{attribute 'linkalways'} 
{attribute 'no_explicit_call' := 'This FB is a CLASS and must be accessed using methods or properties'}
{attribute 'enable_dynamic_creation'}
FUNCTION_BLOCK _TcVnVector2_UINT EXTENDS AliasDatatypeBase
VAR
	localData : TcVnVector2_UINT;
	activeData : REFERENCE TO TcVnVector2_UINT REF= localData;
	aliasBaseDatatype : _Array0to1OfUINT;
END_VAR

PROPERTY PUBLIC Address : PVOID
GET
Address := ADR(activeData);
END_GET
END_PROPERTY

METHOD PUBLIC ClearReference
VAR_INPUT
END_VAR
activeData REF= localData;
SetBaseDatatypeReference();
END_METHOD

METHOD PUBLIC Clone : I_Datatype
VAR
    pClone : POINTER TO _TcVnVector2_UINT;
END_VAR
pClone := __NEW(_TcVnVector2_UINT);
Clone := pClone^;
END_METHOD

METHOD FB_init : BOOL
VAR_INPUT
	bInitRetains : BOOL; // if TRUE, the retain variables are initialized (warm start / cold start)
	bInCopyCode : BOOL;  // if TRUE, the instance afterwards gets moved into the copy code (online change)
	//InitialValue : <type>; // if possible, not all values can be initialized
END_VAR
//localData := InitialValue; // if possible, not all values can be initialized
SetBaseDatatypeReference();
AddBaseDatatype(aliasBaseDatatype);
END_METHOD

PROPERTY PUBLIC Identifier : T_MAXSTRING
GET
Identifier := 'TcVnVector2_UINT';
END_GET
END_PROPERTY

METHOD PUBLIC MakeReferenceTo
VAR_INPUT
	ReferenceTarget : REFERENCE TO TcVnVector2_UINT;
END_VAR
activeData REF= ReferenceTarget;
SetBaseDatatypeReference();
END_METHOD

METHOD PROTECTED SetBaseDatatypeReference
VAR_INPUT
END_VAR
aliasBaseDatatype.MakeReferenceTo(activeData);
END_METHOD

PROPERTY PUBLIC Size : UDINT
GET
Size := SIZEOF(activeData);
END_GET
END_PROPERTY

METHOD TryMakeReferenceTo : BOOL
VAR_INPUT
	Target : I_Datatype;
END_VAR
VAR
	pTargetData : POINTER TO TcVnVector2_UINT;
END_VAR
IF NOT IsEquivalentTo(Target) THEN
	RETURN;
END_IF

pTargetData := Target.Address;
activeData REF= pTargetData^;
SetBaseDatatypeReference();
TryMakeReferenceTo := TRUE;
END_METHOD

PROPERTY PUBLIC Value : REFERENCE TO TcVnVector2_UINT
GET
Value REF= activeData;
END_GET
END_PROPERTY

END_FUNCTION_BLOCK

(* stored: Version 1.1.0.1, ProductVersion 3.1.4024.13
   POU _TcVnVector2_UINT: Id {8bdec0e3-bc1d-03c1-31a8-aad19038b9a6}, SpecialFunc None
   Folder Core: Id {6b5e70ee-943d-0e8f-172c-51f2530f36c3}
   Folder Protected: Id {119f0d77-7c6b-089f-3a92-8e4dc8a1e82c}
   Folder Customize: Id {2d9d9cb3-6aec-0103-3f2c-dbef9294f431}
   Folder Constructor: Id {b36db007-e1b4-09c8-3b4e-b2e25a026cdd}
   Property Address: Id {c7b53c4b-605e-023e-10d5-557ec838859c}
   Get Get: Id {49054a72-2fb9-0ae5-0596-e08a99fd6499}
   Method ClearReference: Id {d99ee36c-9a80-0bea-3cbb-74eb4044bb10}
   Method Clone: Id {a2ad3e3f-6e95-0248-2ab9-1a442c93d6a0}
   Method FB_init: Id {d611d6af-0db9-04e7-3498-a760101e93c0}
   Property Identifier: Id {3a3967f7-87bd-0bda-03e4-1cfae8c89820}
   Get Get: Id {5827e7b2-4da7-0811-0133-1609d0857db7}
   Method MakeReferenceTo: Id {ba81b495-4579-0539-2bb4-f95c47fc08c0}
   Method SetBaseDatatypeReference: Id {9d97bfd3-5923-0244-0fef-217f242ecf3a}
   Property Size: Id {39fd4ca6-5d8e-0667-3dfc-2874494c97f2}
   Get Get: Id {817a9393-a6b9-0b2f-3eb7-53378df1b266}
   Method TryMakeReferenceTo: Id {cc06b6df-3987-0f7f-2523-1589e37c06aa}
   Property Value: Id {5ea25478-eb5b-0fc7-36eb-2fe1836e8542}
   Get Get: Id {ada9b1b1-34af-0455-1366-3f3e113f929e} *)
